//{attribute 'hide_all_locals'}
FUNCTION_BLOCK FB_TcpSendReceivingQueue
VAR_INPUT
	bEnable 			: BOOL; 							//启用
	bReset 				: BOOL; 							//复位,目前设置了自动重连,所以该输入没实现
	sRemoteIp 			: T_IPv4Addr; 						//目标Ip
	nRemotePort 		: UDINT; 							//目标端口
	pRecvData 			: POINTER TO BYTE; 					//接收地址
	nRecvSize 			: UDINT; 							//接收数据区域大小
END_VAR
VAR_OUTPUT
	bBusyConnect 	: BOOL; 								//连接中
	bConnected 		: BOOL; 								//连接完成
	bBusySend 		: BOOL; 								//发送中
	bSendDone 		: BOOL; 								//发送完成
	bBusyRecv 		: BOOL; 								//接受中
	bRecvDone 		: BOOL; 								//接收完成
	bError 			: BOOL; 								//报错
	nRecvBytes 		: UDINT; 								//接收数据长度
	bDataReceived 	: BOOL; 								//接收到数据
END_VAR
VAR
	//功能块调用
	fbConnect : FB_SocketConnect;
	fbClose : FB_SocketClose;
	fbSend : FB_SocketSend;
	fbRecv : FB_SocketReceive;
	fbQueue : FB_SimpleTcpTaskQueue2;
	CurrentTask : ST_TcpTask2;
	//状态流转
	stepSendRecv :UDINT;
	stepReceiving : UDINT;
	stepSend : UDINT;
	//连接部分
	tonReconnect : TON;
	hSocket : T_HSOCKET;
	
	//数据收发
	tonRecv : TON;
	tempData : ARRAY[0..MAXBUFFERSIZE] OF BYTE;
	hr: HRESULT;
	nCountRecvErr : UDINT;

END_VAR

VAR CONSTANT
	MAXBUFFERSIZE: DINT := 1023;
	EmptyhSocket : T_HSOCKET := (handle := 0);
END_VAR

IF pRecvData = 0  THEN
	RETURN;
END_IF
//主逻辑
_CyclicLogic();

METHOD PROTECTED _CyclicLogic : BOOL
VAR_INPUT
END_VAR

VAR
END_VAR
fbQueue();
CurrentTask := fbQueue.CurrentTask;
tonReconnect(IN:= , PT:= T#3S, Q=> , ET=> );
bBusyConnect := (stepSendRecv <> 20);
bConnected := (stepSendRecv = 20);
bError := fbConnect.bError OR fbClose.bError OR fbSend.bError OR fbRecv.bError;

CASE stepSendRecv OF
	0: //初始状态，等待TCP连接
	fbConnect(bExecute:= FALSE);
	fbClose(bExecute:= FALSE);
	fbSend(bExecute:= FALSE);
	fbRecv(bExecute := FALSE);
	tonReconnect.IN := FALSE;
	nCountRecvErr := 0;
	IF bEnable AND sRemoteIp <> '' AND nRemotePort <> 0 THEN
		stepSendRecv := 10;
	END_IF

	10: //连接中
	fbConnect(sRemoteHost:= sRemoteIp, nRemotePort:= nRemotePort, bExecute:= TRUE);
	IF fbConnect.bBusy THEN
		;
	ELSE
		IF NOT fbConnect.bError AND (fbConnect.hSocket.handle <> 0) THEN
			hSocket := fbConnect.hSocket;
			stepSendRecv := 20;
		ELSE
			stepSendRecv := 12;
		END_IF
	END_IF

	12: //重连等待
	tonReconnect.IN := TRUE;
	IF tonReconnect.Q THEN
		stepSendRecv := 0;
		tonReconnect.IN := FALSE;
	END_IF

	20: //连接完成
	_Send();
	hr := _Receiving(200,5); // 接收间隔200ms, 报错限制5次
	IF FAILED(hr) THEN
		stepSendRecv := 30;
	END_IF
	
	
	30:
	fbClose(hSocket:= hSocket, bExecute:= TRUE );
	IF fbClose.bBusy THEN
		;
	ELSE
		hSocket := EmptyhSocket;
		stepSendRecv := 0;
	END_IF
END_CASE
END_METHOD

METHOD PROTECTED _Receiving : HRESULT
VAR_INPUT
	CycleTime : UDINT;
	ErrorLimit : UDINT;
END_VAR
tonRecv(IN:= , PT:= UDINT_TO_TIME(CycleTime), Q=> , ET=> );
bBusyRecv := (stepReceiving = 10 );
bRecvDone := (stepReceiving <> 10 );
CASE stepReceiving OF
	0:
	bDataReceived := FALSE;
	tonRecv.IN := FALSE;
	fbRecv(bExecute := FALSE);
	stepReceiving := 10;
	
	10:
	
	fbRecv(hSocket:= hSocket, cbLen:= SIZEOF(tempData), pDest:= ADR(tempData), bExecute:= TRUE);
	IF fbRecv.bBusy THEN
		;
	ELSE
		IF fbRecv.bError THEN
			nCountRecvErr := nCountRecvErr + 1;
			IF (nCountRecvErr > ErrorLimit) THEN
				_Receiving := -1;
			END_IF
			
		ELSE
			nCountRecvErr := 0;
			IF fbRecv.nRecBytes <> 0 THEN
				MEMSET(destAddr:= pRecvData, fillByte:= 0, n:= nRecvSize);
				MEMCPY(destAddr:= pRecvData, srcAddr:= ADR(tempData), n:= MIN(fbRecv.nRecBytes,nRecvSize) );
				bDataReceived := TRUE;
			END_IF
			nRecvBytes := fbRecv.nRecBytes;
		END_IF
		stepReceiving := 20;
		tonRecv.IN := TRUE;
	END_IF

	20:
	
	tonRecv.IN := TRUE;
	IF tonRecv.Q THEN
		tonRecv.IN := FALSE;
		stepReceiving := 0;
	END_IF

END_CASE
END_METHOD

METHOD PROTECTED _Send : BOOL
VAR_INPUT
END_VAR
bBusySend := (stepSend <> 0);
bSendDone := (stepSend = 0);
CASE stepSend OF
	0:
	fbSend(bExecute:= FALSE);
	IF fbQueue.ActingTaskCount <> 0 THEN
		stepSend := 10;
	END_IF
	
	
	10:
	fbSend(hSocket:= hSocket, cbLen:= CurrentTask.nData, pSrc:= CurrentTask.pData, bExecute:= TRUE);
	IF fbSend.bBusy THEN
		;
	ELSE
		IF fbSend.bError THEN
			_Send := TRUE;
		ELSE
			;
		END_IF
		stepSend := 0;
		fbQueue.FinishTask();
	END_IF
END_CASE
END_METHOD

METHOD AddTask : BOOL
VAR_INPUT
	TaskName : STRING(24);
	TaskType : INT; (* 0:Once, 1:Regular *)
	pData : PVOID;
	nData : UDINT;
END_VAR
fbQueue.AddActingTask(TaskName, TaskType, pData, nData);
END_METHOD

END_FUNCTION_BLOCK

(* stored: Version 1.1.0.1, ProductVersion 3.1.4024.12
   POU FB_TcpSendReceivingQueue: Id {b125606c-342d-446d-9273-736d49487372}, SpecialFunc None
   Method _CyclicLogic: Id {afb564a5-21bf-44d9-be86-fa2e04e17b89}
   Method _Receiving: Id {e9da7ff7-d241-4e1e-8025-1d884b397d9b}
   Method _Send: Id {303f95f9-99be-428d-b1f4-85ee86ac10e3}
   Method AddTask: Id {74e7648e-1c58-4301-81bc-c10ed9d8c3e5} *)
